KUKA KRL data list: $config.dat

&ACCESS RV$5
DEFDAT $CONFIG

ENDDAT
